(* IEC 61131-3 sources: LabBench/Глобальные переменные, 4 files *)

(* ---- GVL_DiagSystem.st ---- *)
(*==============================================================================
    Название:    GVL_DiagSystem_Extended
    Автор:
    Дата:        2025-04-30
    Версия:      1.0

    Описание:    Глобальные переменные расширенной диагностической системы
==============================================================================*)
VAR_GLOBAL CONSTANT
    (* Количество ошибок и сценариев в системе *)
    MAX_ERRORS: UINT := 50;                  (* Максимальное количество ошибок *)
    MAX_SCENARIOS: UINT := 25;               (* Максимальное количество сценариев *)

    (* Идентификаторы систем *)
    SYSTEM_ID: WORD := 16#0100;              (* Общесистемные ошибки *)
    MEASUREMENT_ID: WORD := 16#0200;         (* Ошибки системы измерения *)
    EQUIPMENT_ID: WORD := 16#0300;           (* Ошибки оборудования *)
    COMMUNICATION_ID: WORD := 16#0400;       (* Ошибки связи *)

    (* Идентификаторы подсистем измерения *)
    PRESSURE_SENSORS_ID: WORD := 16#0210;    (* Датчики давления *)
    LEVEL_SENSORS_ID: WORD := 16#0220;       (* Датчики уровня *)
    FLOW_SENSORS_ID: WORD := 16#0230;        (* Расходомеры *)
    TEMP_SENSORS_ID: WORD := 16#0240;        (* Датчики температуры *)

    (* Идентификаторы оборудования *)
    PROP_VALVE_ID: WORD := 16#0310;          (* Пропорциональный клапан *)
    EM_VALVE_ID: WORD := 16#0320;            (* Электромагнитный клапан *)
    PUMP1_ID: WORD := 16#0330;               (* Насос 1 *)
    PUMP2_ID: WORD := 16#0340;               (* Насос 2 *)
    HEATER_ID: WORD := 16#0350;              (* Нагреватель (ТЭН) *)

    (* Идентификаторы связи *)
    SCADA_COMM_ID: WORD := 16#0410;          (* Связь со SCADA *)
    MODBUS_COMM_ID: WORD := 16#0420;         (* Связь по Modbus (ТРМ10) *)
END_VAR

VAR_GLOBAL
    (* Массивы ошибок и сценариев *)
    gaBlockingErrors: ARRAY[1..MAX_ERRORS] OF ST_BlockingError;     (* Массив ошибок *)
    gaDiagScenarios: ARRAY[1..MAX_SCENARIOS] OF ST_DiagScenario;    (* Массив сценариев *)

    (* Состояние системы *)
    geSystemState: E_SystemState;            (* Текущее состояние системы *)
    gxSystemBlockingRequired: BOOL;          (* Требуется блокировка системы *)
    gxSystemShutdownRequired: BOOL;          (* Требуется останов системы *)
    gxSystemResetRequired: BOOL;             (* Требуется сброс системы *)
    gstShutdownSequence: ST_ShutdownSequence;(* Последовательность останова *)

    (* Агрегированная информация о сценариях *)
    gxAnyScenarioActive: BOOL;               (* Любой сценарий активен *)
    gxAnyScenarioBlockingRequired: BOOL;     (* Любой сценарий требует блокировки *)
    gxAnyScenarioShutdownRequired: BOOL;     (* Любой сценарий требует останова *)
    gdwActiveScenariosMask: DWORD;           (* Битовая маска активных сценариев *)
    giLastActiveScenarioIndex: UINT;         (* Индекс последнего активного сценария *)

    (* Агрегированные состояния *)
    gxAnyError: BOOL;                        (* Флаг наличия любых ошибок *)
    gxSystemBlocking: BOOL;                  (* Флаг полной блокировки системы *)
    gdwActiveErrorMask: DWORD;               (* Битовая маска активных ошибок *)

    (* Блокировки устройств *)
    gxPropValveBlocking: BOOL;               (* Блокировка пропорционального клапана *)
    gxEMValveBlocking: BOOL;                 (* Блокировка электромагнитного клапана *)
    gxPump1Blocking: BOOL;                   (* Блокировка насоса 1 *)
    gxPump2Blocking: BOOL;                   (* Блокировка насоса 2 *)
    gxHeaterBlocking: BOOL;                  (* Блокировка нагревателя *)

    (* Управление лампой *)
    geLampMode: E_LampBlinkMode;             (* Режим работы сигнальной лампы *)
    gxLampState: BOOL;                       (* Текущее состояние лампы *)

    (* Команды управления *)
    gxResetAll: BOOL;                        (* Сброс всех ошибок *)
    gxResetMeasurement: BOOL;                (* Сброс ошибок измерительной системы *)
    gxResetPropValve: BOOL;                  (* Сброс ошибок пропорционального клапана *)
    gxResetEMValve: BOOL;                    (* Сброс ошибок электромагнитного клапана *)
    gxResetPump1: BOOL;                      (* Сброс ошибок насоса 1 *)
    gxResetPump2: BOOL;                      (* Сброс ошибок насоса 2 *)
    gxResetHeater: BOOL;                     (* Сброс ошибок нагревателя *)
    gxStartNormalShutdown: BOOL;             (* Запуск нормального останова *)
    gxStartEmergencyShutdown: BOOL;          (* Запуск аварийного останова *)
END_VAR

(* ---- GVL_Equipments.st ---- *)
(*==============================================================================
    Название:    GVL_Equipments
    Автор:       Редько А.
    Дата:        2025-04-27
    Версия:      1.0

    Описание:    Глобальные переменные оборудования
==============================================================================*)
VAR_GLOBAL
    (* Структуры данных оборудования *)
    stPropValve: ST_PropValve;       (* Пропорциональный кран *)
END_VAR

(* ---- GVL_Inputs.st ---- *)
(*==============================================================================
    Название:    GVL_WaterSystem
    Автор:       Редько А.
    Дата:        2025-04-23
    Версия:      1.0

    Описание:    Глобальные переменные системы датчиков
==============================================================================*)
VAR_GLOBAL
    GVL_stHydroLevel_KIE1: 		ST_HydroLevel_Data;     	(* Структура гидростатического датчика уровня в емкости КИЕ1 *)
    GVL_stPressureKIE2: 		ST_PressureSensor_Data;		(* Структура датчика давления в емкости КИЕ2 *)
    GVL_stPressurePipe: 		ST_PressureSensor_Data;   	(* Структура датчика давления в трубопроводе *)
    GVL_stPressurePumpIn1:		ST_PressureSensor_Data;  	(* Структура датчика давления перед насосом 1 *)
    GVL_stPressurePumpOut1:     ST_PressureSensor_Data;  	(* Структура датчика давления после насоса 1 *)
    GVL_stPressurePumpIn2: 		ST_PressureSensor_Data;  	(* Структура датчика давления перед насосом 2 *)
    GVL_stPressurePumpOut2: 	ST_PressureSensor_Data;  	(* Структура датчика давления после насоса 2 *)
    GVL_stFloatLevelSensors:    ST_FloatLevelGroup_Data;    (* Структура группы поплавковых датчиков уровня *)
END_VAR

(* ---- GVL_SCADA.st ---- *)
(*==============================================================================
    Название:    GVL_SCADA
    Автор:       Редько А.
    Дата:        2025-04-27
    Версия:      1.0

    Описание:    Глобальные переменные для интерфейса SCADA
==============================================================================*)
VAR_GLOBAL
    (* Пропорциональный кран - входные переменные (из SCADA в ПЛК) *)
    GVL_in_SCADA_PropValve_Mode: E_EquipmentMode := MANUAL;    (* Режим работы *)
    GVL_in_SCADA_PropValve_SetPosition: REAL := 0.0;           (* Задание положения (0-100%) *)
    GVL_in_SCADA_PropValve_Reset: BOOL := FALSE;               (* Сброс ошибок *)
    GVL_in_SCADA_PropValve_SafePosition: REAL := 0.0;          (* Безопасное положение (0-100%) - закрыт *)

    (* Пропорциональный кран - выходные переменные (из ПЛК в SCADA) *)
    GVL_out_SCADA_PropValve_ActualPosition: REAL;              (* Текущее положение (0-100%) *)
    GVL_out_SCADA_PropValve_TargetPosition: REAL;              (* Целевое положение (0-100%) *)
    GVL_out_SCADA_PropValve_Mode: E_EquipmentMode;             (* Текущий режим работы *)
    GVL_out_SCADA_PropValve_State: E_PropValveState;           (* Состояние крана *)
    GVL_out_SCADA_PropValve_ErrorCode: WORD;                   (* Код ошибки *)
    GVL_out_SCADA_PropValve_Moving: BOOL;                      (* Флаг движения крана *)

    (* Электромагнитный клапан - входные переменные (из SCADA в ПЛК) *)
    GVL_in_SCADA_EMValve_Open: BOOL := FALSE;                (* Команда открытия *)
    GVL_in_SCADA_EMValve_Reset: BOOL := FALSE;               (* Сброс счетчиков *)
    GVL_in_SCADA_EMValve_WarningTime: TIME := T#15M;         (* Порог предупреждения *)

    (* Электромагнитный клапан - выходные переменные (из ПЛК в SCADA) *)
    GVL_out_SCADA_EMValve_IsOpen: BOOL;                      (* Текущее состояние *)
    GVL_out_SCADA_EMValve_State: E_EMValveState;             (* Состояние клапана *)
    GVL_out_SCADA_EMValve_ContinuousOpTime: TIME;            (* Время непрерывной работы *)
    GVL_out_SCADA_EMValve_TotalOpTime: TIME;                 (* Общее время работы *)
END_VAR
